FUNCTION_BLOCK FINAL FB_Statistics
VAR_INPUT
	Description				: STRING(31);			//Statistic description
	Trigger					: BOOL;					//New item trigger
	PerPulse				: REAL;					//Items per pulse
END_VAR
VAR
	_Reset					: BOOL;					//Reset Statistics
	_CycleTime				: REAL;					//Time for one item cycle (seconds)
	_CurrentRate			: REAL;					//Current item rate per minute
	_ThisMin				: REAL;					//Number of items processed this minute
	_LastMin				: REAL;					//Number of items processed last minute
	_ThisHour				: REAL;					//Number of items processed this hour
	_LastHour				: REAL;					//Number of items processed last hour
	_HistoryAvg				: REAL;					//Average items/minute for the previous 10 minutes
	_History				: ARRAY[1..10] OF REAL; //Item 10minute history
	_InstHistory			: ARRAY[1..20] OF REAL;	//Item instantaneous history
	_ItemCycleTime			: REAL;					//Item cycle time
	_InstHistoryCount		: INT;					//Instantaneous history For loop counter
	_HistoryCount			: INT;					//History For loop counter
	_HistorySum				: REAL;					//History summation holder
	_R_Trig					: R_TRIG;				//Statistic Count Trigger	
	_SecondsCount			: INT;					//Seconds history for loop counter
	_ThisSec				: INT;					//Item count this second
	_SecondsHistory			: ARRAY [0..59] OF INT; //Seconds history
	_ItemsLast60s			: INT;					//Current item rate for last 60 seconds
END_VAR
VAR_IN_OUT
	Control					: ST_System;			//Machine control system time
END_VAR
VAR PERSISTENT
	_LifeTime				: REAL;					//Life time count
	_Today					: REAL;					//Tadays count
END_VAR

//Statistic Count Trigger
_R_Trig	(CLK:=Trigger);

//Total Counts
IF Control.SystemTime.MidnightPulse OR _Reset THEN
	_Today := 0;
ELSE 
	IF _R_Trig.Q THEN
		_LifeTime := _LifeTime + PerPulse;
		_Today := _Today + PerPulse;
		_ThisHour := _ThisHour + PerPulse;
		_ThisMin := _ThisMin + PerPulse;
	END_IF
END_IF

//Cycle Time
IF _R_Trig.Q AND _ItemCycleTime > 0 THEN
	_CycleTime := _ItemCycleTime;
	_CurrentRate := PerPulse * (60 / F_CheckDivReal(_ItemCycleTime));
	_ItemCycleTime := 0;
	FOR _InstHistoryCount := 20 TO 2 BY -1 DO
		_InstHistory[F_CheckIndexBounds(1,10,_InstHistoryCount)] := _InstHistory[F_CheckIndexBounds(1,10,_InstHistoryCount)-1];
	END_FOR
	_InstHistory[1] := _CycleTime;	
ELSIF Control.PackMLState.Execute OR Control.PackMLState.Holding OR Control.PackMLState.UnHolding OR Control.PackMLState.Suspending OR Control.PackMLState.UnSuspending OR Control.PackMLState.Completing  THEN
	_ItemCycleTime := _ItemCycleTime + Control.SystemTime.ScanTime;
END_IF

//Minute Counts and History
IF Control.SystemTime.MinutePulse THEN
	_LastMin := _ThisMin;
	_ThisMin := 0;
	_HistorySum := 0;
	FOR _HistoryCount := 10 TO 2 BY -1 DO
		_History[F_CheckIndexBounds(1,10,_HistoryCount)] := _History[F_CheckIndexBounds(1,10,_HistoryCount)-1];
		_HistorySum := _HistorySum + _History[F_CheckIndexBounds(1,10,_HistoryCount)];
	END_FOR
	_History[1] := _LastMin;
	_HistorySum := _HistorySum + _History[1];
	_HistoryAvg := _HistorySum/10;
END_IF

//Hour counts
IF Control.SystemTime.HourPulse THEN
	_LastHour := _ThisHour;
	_ThisHour := 0;
END_IF

//Seconds Count and History
IF _R_Trig.Q THEN
	_SecondsHistory[_ThisSec] := _SecondsHistory[_ThisSec] + REAL_TO_INT(PerPulse);
END_IF

_ItemsLast60s := 0;
FOR _SecondsCount:= 0 TO 59 DO
	_ItemsLast60s := _ItemsLast60s + _SecondsHistory[_SecondsCount];
END_FOR

IF Control.SystemTime.SecondPulse THEN
	_ThisSec := _ThisSec + 1;
	IF _ThisSec >= 60 THEN _ThisSec := 0; END_IF;
	_SecondsHistory[_ThisSec] := 0;
END_IF

{attribute 'monitoring' := 'variable'}
PROPERTY PUBLIC CurrentRate : REAL
GET
CurrentRate := _CurrentRate;
END_GET
END_PROPERTY

{attribute 'monitoring' := 'variable'}
PROPERTY PUBLIC CycleTime : REAL
GET
CycleTime := _CycleTime;
END_GET
END_PROPERTY

{attribute 'monitoring' := 'variable'}
PROPERTY PUBLIC History : ARRAY[1..10] OF REAL
GET
History := _History;
END_GET
END_PROPERTY

{attribute 'monitoring' := 'variable'}
PROPERTY PUBLIC HistoryAvg : REAL
GET
HistoryAvg := _HistoryAvg;
END_GET
END_PROPERTY

{attribute 'monitoring' := 'variable'}
PROPERTY PUBLIC InstHistory : ARRAY[1..20] OF REAL
GET
InstHistory := _InstHistory;
END_GET
END_PROPERTY

{attribute 'monitoring' := 'variable'}
PROPERTY PUBLIC LastHour : REAL
GET
LastHour := _LastHour;
END_GET
END_PROPERTY

{attribute 'monitoring' := 'variable'}
PROPERTY PUBLIC LastMin : REAL
GET // PUBLIC
LastMin := _LastMin;
END_GET
END_PROPERTY

{attribute 'monitoring' := 'variable'}
PROPERTY PUBLIC Reset : BOOL
GET
Reset := _Reset;
END_GET
SET
_Reset := Reset;
END_SET
END_PROPERTY

{attribute 'monitoring' := 'variable'}
PROPERTY PUBLIC ThisHour : REAL
GET
ThisHour := _ThisHour;
END_GET
END_PROPERTY

{attribute 'monitoring' := 'variable'}
PROPERTY PUBLIC ThisMin : REAL
GET
ThisMin := _ThisMin;
END_GET
END_PROPERTY

END_FUNCTION_BLOCK

(* stored: Version 1.1.0.1, ProductVersion 3.1.4024.3
   POU FB_Statistics: Id {4d66ba82-e7a4-4ed9-a000-21de436fb4b9}, SpecialFunc None
   Property CurrentRate: Id {f8e2e6df-a606-46e3-ac1b-969d9cadd38b}
   Get Get: Id {61880ab1-a8bd-48b4-af64-bbe1afc0b6df}
   Property CycleTime: Id {5f44376c-338f-413e-beb1-acf443b1da5d}
   Get Get: Id {1e7edb77-02c9-469e-9709-90a8e872c67c}
   Property History: Id {f5567f7d-3dad-4f20-9410-65c1add9fce8}
   Get Get: Id {ad6c6aa2-10ac-43ed-860a-66006935450e}
   Property HistoryAvg: Id {1725eb71-5cbf-414a-a784-8607904992a4}
   Get Get: Id {24d51c51-6faa-423c-93b5-f566ddd77646}
   Property InstHistory: Id {64ff3fa2-bda8-42cb-be69-ee50bc63493a}
   Get Get: Id {57f1ebcb-119f-4d43-ab40-9e6609830287}
   Property LastHour: Id {532d1d2b-7a3e-4d4c-b4d5-0984f45b47a7}
   Get Get: Id {65b86eb5-eedf-4be6-b960-152c2b62cf0b}
   Property LastMin: Id {6f8bee78-47a9-4e80-9529-d50ea8a86859}
   Get Get: Id {4c772052-0dc0-459b-a363-660940f93c79}
   Property Reset: Id {ed0f0a91-08d5-4872-9888-0128419c3e20}
   Get Get: Id {3bb69b12-3be4-407c-ad85-cae702043beb}
   Set Set: Id {92f2845a-578e-42e8-b927-06728fbbeaa8}
   Property ThisHour: Id {41286b01-53c1-452d-8f07-890ae7037a8d}
   Get Get: Id {a9641f2f-e280-4aec-8875-864449827aed}
   Property ThisMin: Id {27b685a2-4b2b-47c9-8ece-ac9513cc439b}
   Get Get: Id {e18fd340-700c-465c-85a4-a39cf9a07e43} *)
